(* Logix 5000 project; controller TrayLoader_EnSG vendor 1 type 14 code 156 rev 32.11; software revision 32.02; part 3 of 3 *)
(* tags used below, declared in another part *)
   blink1s : BOOL;
   ons : DINT;
   t1s_tof : TIMER;
   t1s_ton : TIMER;
   Auto : BOOL;
   man_sv_flipperIn : BOOL;
   man_sv_flipperOut : BOOL;
   man_sv_gripper : BOOL;
   Run : BOOL;
   sv_flipperIn : BOOL;
   sv_flipperOut : BOOL;
   sv_gripper : BOOL;
(* MainProgram, continued *)

ROUTINE _20_Misc   (* ladder *)
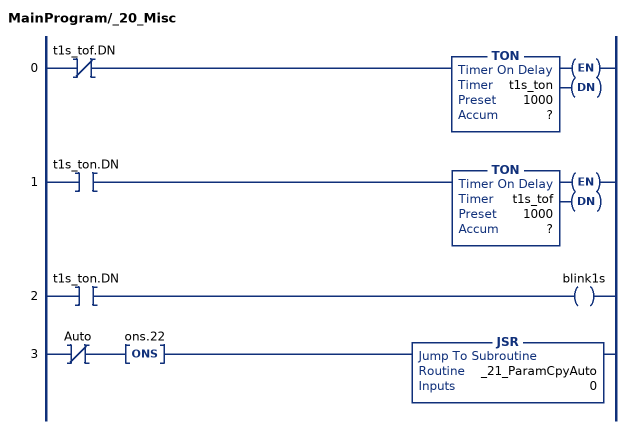
   0: XIO(t1s_tof.DN)TON(t1s_ton,?,?);
   1: XIC(t1s_ton.DN)TON(t1s_tof,?,?);
   2: XIC(t1s_ton.DN)OTE(blink1s);
   3: XIO(Auto)ONS(ons.22)JSR(_21_ParamCpyAuto,0);
END_ROUTINE

ROUTINE _21_ParamCpyAuto   (* structured text *)
   (* To transfer states from Auto to Manual Mode, so that, during mode switching, no changes in states,
   for example for gripper, if in auto mode, the state is grip, but in manual mode it has release state, the tray will drop
   *)
   man_sv_flipperIn := sv_flipperIn;
   man_sv_flipperOut := sv_flipperOut;
   man_sv_gripper := sv_gripper;
   
   
END_ROUTINE

ROUTINE MainRoutine   (* ladder *)
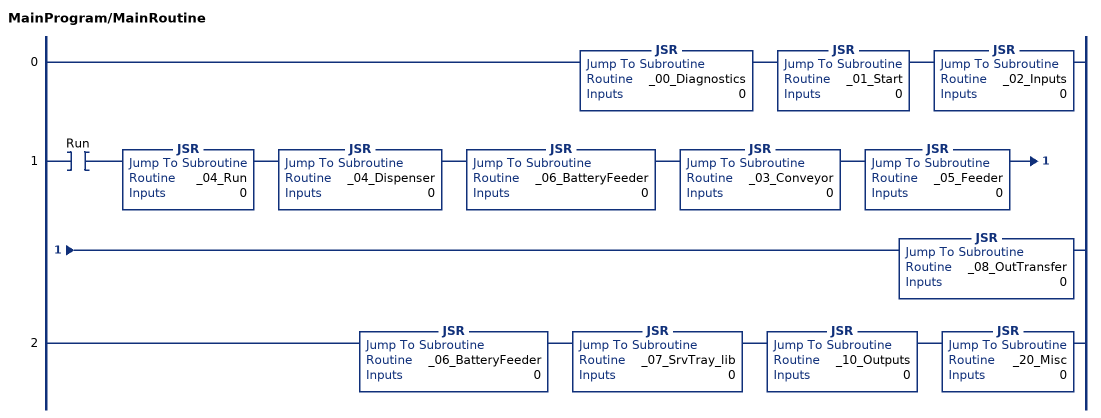
   0: JSR(_00_Diagnostics,0)JSR(_01_Start,0)JSR(_02_Inputs,0);
   1: XIC(Run)JSR(_04_Run,0)JSR(_04_Dispenser,0)JSR(_06_BatteryFeeder,0)JSR(_03_Conveyor,0)JSR(_05_Feeder,0)JSR(_08_OutTransfer,0);
   2: JSR(_06_BatteryFeeder,0)JSR(_07_SrvTray_lib,0)JSR(_10_Outputs,0)JSR(_20_Misc,0);
END_ROUTINE
END_PROGRAM
